// TIA Portal V15.1 export
// export: Created 2024-06-21T08:41:00.513514Z, ExportSetting WithDefaults, DisplayName Totally Integrated Automation Portal, DisplayVersion V15.1 Update 5, DisplayName TIA Portal Openness, DisplayVersion V15.1 Update 5, DisplayName SINAMICS Startdrive Advanced, DisplayVersion V15.1, DisplayName G130, G150, S120, S150, SINAMICS MV, S210, DisplayVersion V15.1, DisplayName G110M, G120, G120C, G120D, G120P, DisplayVersion V15.1, DisplayName STEP 7 Professional, DisplayVersion V15.1 Update 5, DisplayName STEP 7 Safety, DisplayVersion V15.1, DisplayName WinCC Professional, DisplayVersion V15.1 Update 5, DisplayName SIMATIC Visualization Architect, DisplayVersion V15.1
FUNCTION_BLOCK "LDP/PNCouplerCheck"   // FB1900, FBD
TITLE = LDPCouplerCheck
{ S7_Optimized_Access := 'FALSE' }
AUTHOR : VCC
FAMILY : Communic
NAME : LDPCheck
VERSION : 0.1
// ================================================================================
// This FB checks the communication between 2 plc's via DP/DP coupler
// ================================================================================
// stored: AutoNumber false, IsIECCheckEnabled false, SetENOAutomatically False, UDAEnableTagReadback false
   VAR_INPUT
      I_CheckPlcCom { ExternalAccessible := 'False'; ExternalVisible := 'False'; ExternalWritable := 'False'} : Bool;   // Input from other plc via DP/DP coupler
      I_AlarmResetPB { ExternalAccessible := 'False'; ExternalVisible := 'False'; ExternalWritable := 'False'} : Bool;   // Alarm reset pushbutton is activated
   END_VAR
   VAR_OUTPUT
      O_CheckPlcCom { ExternalAccessible := 'False'; ExternalVisible := 'False'; ExternalWritable := 'False'} : Bool;   // Output to other plc via DP/DP coupler
      O_DPCouplerResponseAlarm { ExternalAccessible := 'False'; ExternalVisible := 'False'; ExternalWritable := 'False'} : Bool;   // Profibus DP coupler alarm
      O_AlarmABCondition { ExternalAccessible := 'False'; ExternalVisible := 'False'; ExternalWritable := 'False'} : Bool;   // Alarm AB condition
      H_IAnim { ExternalAccessible := 'False'; ExternalVisible := 'False'; ExternalWritable := 'False'} : Word;   // Animation
   END_VAR
   VAR DB_SPECIFIC
      H_Out : Struct   // HMI
         Anim : Word;   // HMI Animation of the object
         DBnr : Int;   // HMI Animation DB number
      END_STRUCT;
      DPCouplerResponseAlarm { ExternalAccessible := 'False'; ExternalVisible := 'False'; ExternalWritable := 'False'} : Bool;   // Profibus DP coupler alarm
      ResponseTimeOffAlarm { ExternalAccessible := 'False'; ExternalVisible := 'False'; ExternalWritable := 'False'} : Bool;   // Alarm : signal from other plc stays ON
      ResponseTimeOnAlarm { ExternalAccessible := 'False'; ExternalVisible := 'False'; ExternalWritable := 'False'} : Bool;   // Alarm : signal from other plc stays OFF
      ChangeStatePulse { ExternalAccessible := 'False'; ExternalVisible := 'False'; ExternalWritable := 'False'} : Bool;   // Pulse to change state every 3 sec
      CheckPLC { ExternalAccessible := 'False'; ExternalVisible := 'False'; ExternalWritable := 'False'} : Bool;   // Variable changing from state every 3 sec
      CheckPlcCom { ExternalAccessible := 'False'; ExternalVisible := 'False'; ExternalWritable := 'False'} : Bool;   // Variable changing from state every 3 sec
      ChangeStateTime { ExternalAccessible := 'False'; ExternalVisible := 'False'; ExternalWritable := 'False'} : DInt := DINT#3000;   // Time between 2 pulses
      AlarmResponseTime { ExternalAccessible := 'False'; ExternalVisible := 'False'; ExternalWritable := 'False'} : DInt := DINT#5000;   // Time to create alarm
      DPCouplerResponseAlmCond { ExternalAccessible := 'False'; ExternalVisible := 'False'; ExternalWritable := 'False'} : Bool;   // Profibus DP coupler alarm condition
      DBnr { ExternalAccessible := 'False'; ExternalVisible := 'False'; ExternalWritable := 'False'} : Int;   // HMI DB number
      InputCheckPlcCom { ExternalAccessible := 'False'; ExternalVisible := 'False'; ExternalWritable := 'False'} : Bool;   // Input from other plc via DP/DP coupler
   END_VAR
   VAR
      ResponsTimer1 { ExternalAccessible := 'False'; ExternalVisible := 'False'; ExternalWritable := 'False'; S7_SetPoint := 'True'} : "LTimer";   // Timer to create alarm
      ResponsTimer2 { ExternalAccessible := 'False'; ExternalVisible := 'False'; ExternalWritable := 'False'; S7_SetPoint := 'True'} : "LTimer";   // Timer to create alarm
      StateTimer { ExternalAccessible := 'False'; ExternalVisible := 'False'; ExternalWritable := 'False'; S7_SetPoint := 'True'} : "LTimer";   // Timer to create pulse to change status
   END_VAR
BEGIN

NETWORK
TITLE = **** 1 - Inputs **** DB number
// DB number
      L     DINO;
      T     #DBnr;

REGION Network 2: **** 1 - Inputs **** Input from other plc via DP/DP coupler
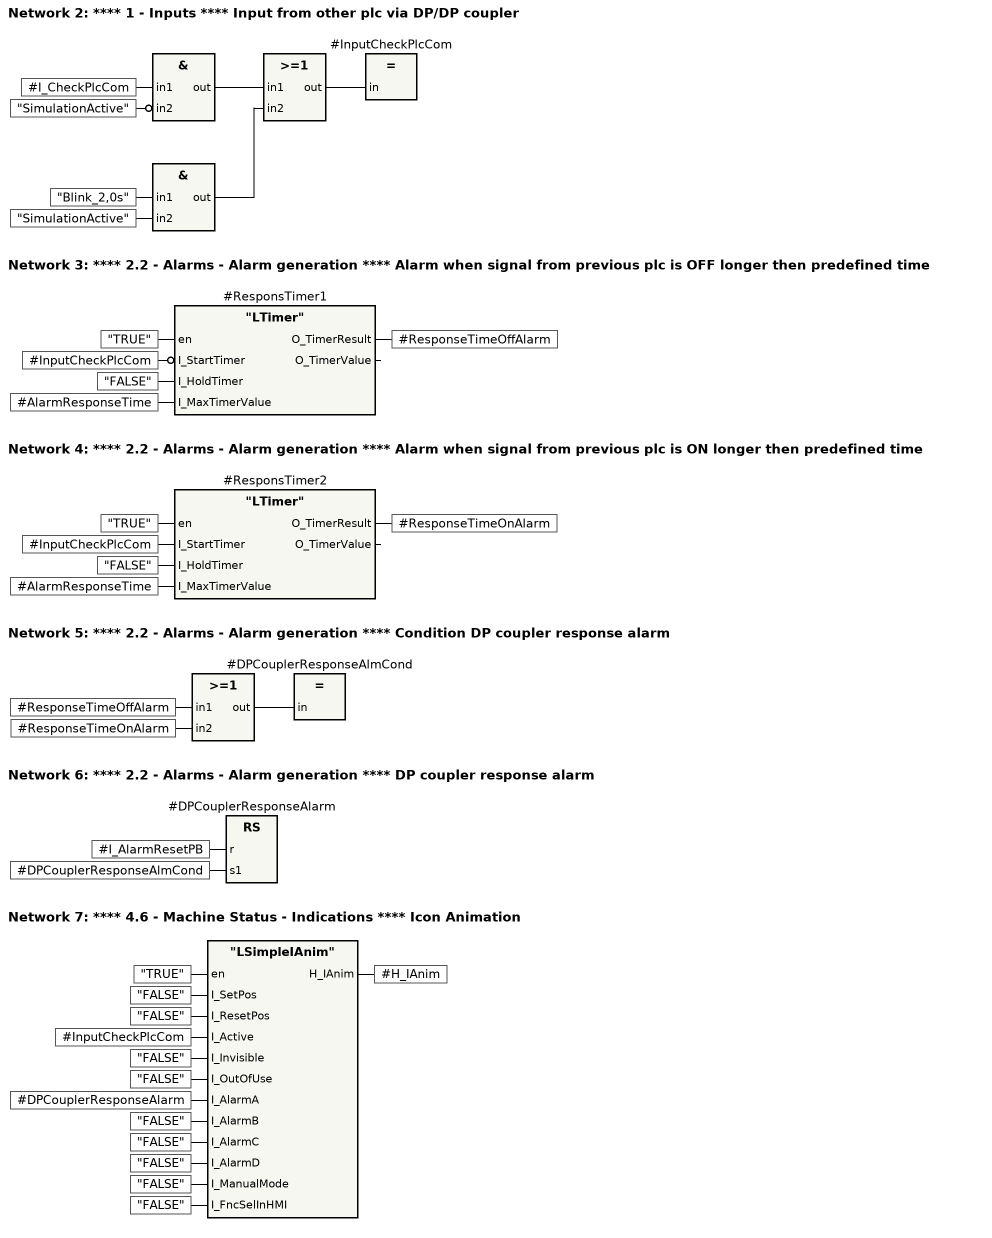
   #InputCheckPlcCom := (#I_CheckPlcCom AND NOT "SimulationActive") OR ("Blink_2,0s" AND "SimulationActive");
END_REGION

REGION Network 3: **** 2.2 - Alarms - Alarm generation **** Alarm when signal from previous plc is OFF longer then predefined time
   // Alarm when signal from previous plc is OFF longer then predefined time
   IF "TRUE" THEN
       #ResponsTimer1(I_StartTimer := NOT #InputCheckPlcCom,   // "LTimer"
                      I_HoldTimer := "FALSE",
                      I_MaxTimerValue := #AlarmResponseTime,
                      O_TimerResult => #ResponseTimeOffAlarm);
   END_IF;
END_REGION

REGION Network 4: **** 2.2 - Alarms - Alarm generation **** Alarm when signal from previous plc is ON longer then predefined time
   // Alarm when signal from previous plc is ON longer then predefined time
   IF "TRUE" THEN
       #ResponsTimer2(I_StartTimer := #InputCheckPlcCom,   // "LTimer"
                      I_HoldTimer := "FALSE",
                      I_MaxTimerValue := #AlarmResponseTime,
                      O_TimerResult => #ResponseTimeOnAlarm);
   END_IF;
END_REGION

REGION Network 5: **** 2.2 - Alarms - Alarm generation **** Condition DP coupler response alarm
   // Condition DP coupler response alarm
   #DPCouplerResponseAlmCond := #ResponseTimeOffAlarm OR #ResponseTimeOnAlarm;
END_REGION

REGION Network 6: **** 2.2 - Alarms - Alarm generation **** DP coupler response alarm
   // DP coupler response alarm
   IF #I_AlarmResetPB THEN
       #DPCouplerResponseAlarm := FALSE;   // RS flip-flop
   END_IF;
   IF #DPCouplerResponseAlmCond THEN #DPCouplerResponseAlarm := TRUE; END_IF;
END_REGION

REGION Network 7: **** 4.6 - Machine Status - Indications **** Icon Animation
   // Icon Animation
   IF "TRUE" THEN
       "LSimpleIAnim"(I_SetPos := "FALSE",
                      I_ResetPos := "FALSE",
                      I_Active := #InputCheckPlcCom,
                      I_Invisible := "FALSE",
                      I_OutOfUse := "FALSE",
                      I_AlarmA := #DPCouplerResponseAlarm,
                      I_AlarmB := "FALSE",
                      I_AlarmC := "FALSE",
                      I_AlarmD := "FALSE",
                      I_ManualMode := "FALSE",
                      I_FncSelInHMI := "FALSE",
                      H_IAnim => #H_IAnim);
   END_IF;
END_REGION

REGION Network 8: **** 4.6 - Machine Status - Indications **** Animation
   // Animation
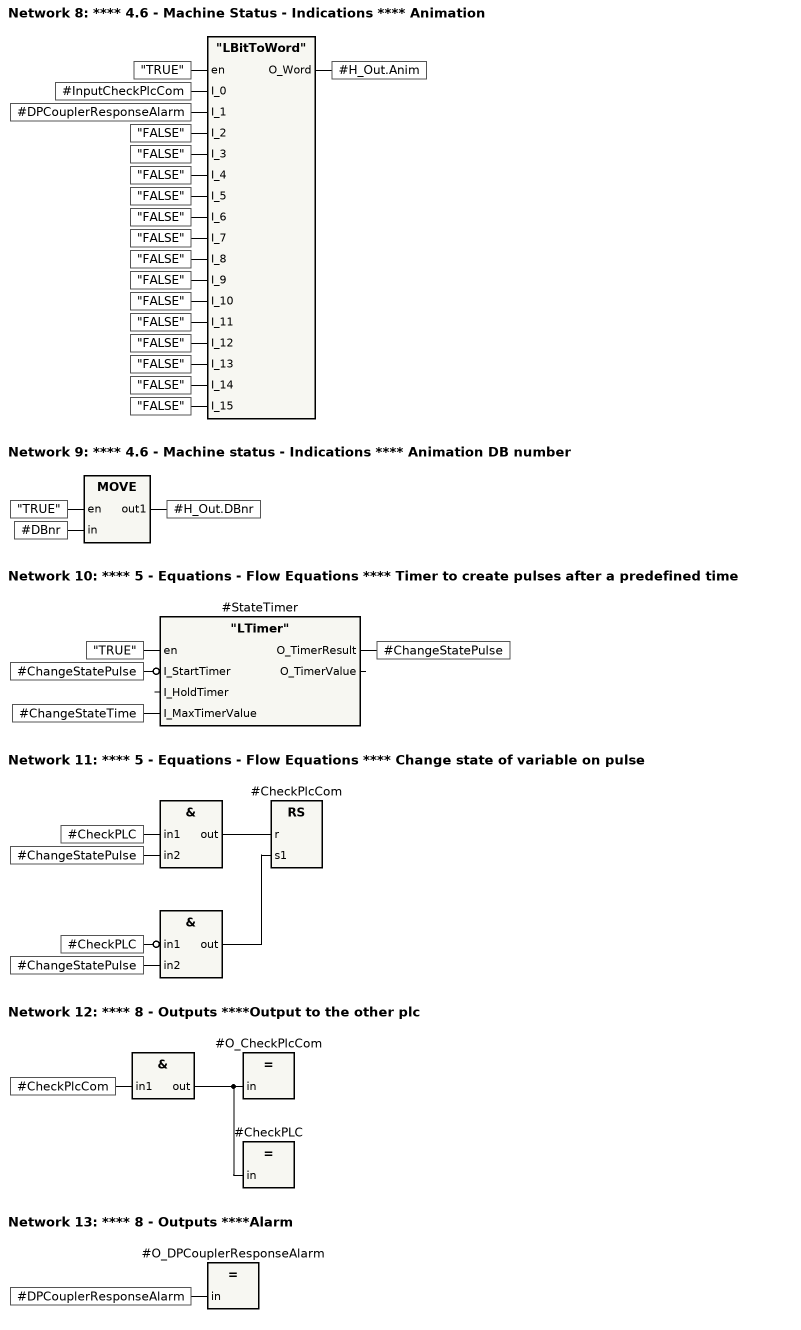
   IF "TRUE" THEN
       "LBitToWord"(I_0 := #InputCheckPlcCom,
                    I_1 := #DPCouplerResponseAlarm,
                    I_2 := "FALSE",
                    I_3 := "FALSE",
                    I_4 := "FALSE",
                    I_5 := "FALSE",
                    I_6 := "FALSE",
                    I_7 := "FALSE",
                    I_8 := "FALSE",
                    I_9 := "FALSE",
                    I_10 := "FALSE",
                    I_11 := "FALSE",
                    I_12 := "FALSE",
                    I_13 := "FALSE",
                    I_14 := "FALSE",
                    I_15 := "FALSE",
                    O_Word => #H_Out.Anim);
   END_IF;
END_REGION

REGION Network 9: **** 4.6 - Machine status - Indications **** Animation DB number
   // Animation DB number
   IF "TRUE" THEN #H_Out.DBnr := #DBnr; END_IF;
END_REGION

REGION Network 10: **** 5 - Equations - Flow Equations **** Timer to create pulses after a predefined time
   // Timer to create pulses after a predefined time
   IF "TRUE" THEN
       #StateTimer(I_StartTimer := NOT #ChangeStatePulse,   // "LTimer"
                   I_MaxTimerValue := #ChangeStateTime,
                   O_TimerResult => #ChangeStatePulse);
   END_IF;
END_REGION

REGION Network 11: **** 5 - Equations - Flow Equations **** Change state of variable on pulse
   // Change state of variable on pulse
   IF #CheckPLC AND #ChangeStatePulse THEN
       #CheckPlcCom := FALSE;   // RS flip-flop
   END_IF;
   IF NOT #CheckPLC AND #ChangeStatePulse THEN #CheckPlcCom := TRUE; END_IF;
END_REGION

REGION Network 12: **** 8 - Outputs ****Output to the other plc
   // Output to the other plc
   #O_CheckPlcCom := #CheckPlcCom;
   #CheckPLC := #CheckPlcCom;
END_REGION

REGION Network 13: **** 8 - Outputs ****Alarm
   // Alarm
   #O_DPCouplerResponseAlarm := #DPCouplerResponseAlarm;
END_REGION

REGION Network 14: **** 8 - Outputs **** Alarm Resetable
   // Alarm Resetable
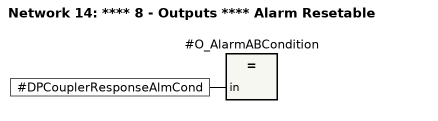
   #O_AlarmABCondition := #DPCouplerResponseAlmCond;
END_REGION
END_FUNCTION_BLOCK
